// TIA Portal project "Sequential Tank Transfer System" (V17)

(* hardware
DEVICE "S7-1500/ET200MP station_1"  S7-1500 station
   slot 0: "Rail_0"  Rack  6ES7 590-1***0-0AA0
   slot 1: "PLC_STTS_01"  CPU 1512C-1 PN  6ES7 512-1CK00-0AB0  V2.9
      slot 3: "CPU display_1"  6ES7591-1AA00-0AA0
      slot 32768: "PROFINET interface_1"  X1
         slot 32769: "Port_1"  X1 P1
         slot 32770: "Port_2"  X1 P2
      slot 34817: "Virtual CP interface port_1"  Virtual CP interface port  Virtual CP interface port
DEVICE "HMI_1"  TP700 Comfort
   slot 0: "HMI_1"  TP700 Comfort  6AV2 124-0GC01-0AX0  17.0.0.0
   slot 1: "HMI_RT_1"  TP700 Comfort  6AV2 124-0GC01-0AX0  17.0.0.0
   slot 5: "HMI_1.IE_CP_1"  PROFINET Interface  17.0.0.0
      slot 1: "PROFINET Interface_1"  PROFINET Interface
         slot 1: "Port_1"  Port
         slot 2: "Port_2"  Port
   slot 7: "HMI_1.MPI/DP_CP_1"  MPI/DP Interface  17.0.0.0
*)

// ===== PLC "PLC_STTS_01"  CPU 1512C-1 PN =====

VAR_GLOBAL   // PLC tag table "STTS_Table"
   "PB_Start" AT %I10.0 : Bool;   // Begins the sequence
   "PB_Stop" AT %I10.1 : Bool;   // Emergency stop function
   "Max_Lvl_T1" AT %I10.2 : Bool;   // Indicates when Tank 1 is full
   "Min_Lvl_T1" AT %I10.3 : Bool;   // Indicates when Tank 1 is empty
   "Max_Lvl_T2" AT %I10.4 : Bool;   // Indicates when Tank 2 is full
   "Min_Lvl_T2" AT %I10.5 : Bool;   // Indicates when Tank 2 is empty
   "Is_Open_V1" AT %I10.6 : Bool;   // Confirmation that Valve 1 is fully open
   "Is_Closed_V1" AT %I10.7 : Bool;   // Confirmation that Valve 1 is fully closed
   "Is_Open_V2" AT %I11.0 : Bool;   // Confirmation that Valve 2 is fully open
   "Is_Closed_V2" AT %I11.1 : Bool;   // Confirmation that Valve 2 is fully closed
   "Is_Open_V3" AT %I11.2 : Bool;   // Confirmation that Valve 3 is fully open
   "Is_Closed_V3" AT %I11.3 : Bool;   // Confirmation that Valve 3 is fully closed
   "Is_Open_V4" AT %I11.4 : Bool;   // Confirmation that Valve 4 is fully open
   "Is_Closed_V4" AT %I11.5 : Bool;   // Confirmation that Valve 4 is fully closed
   "FBK_P2" AT %I11.6 : Bool;   // Running feedback from Pump 2
   "FBK_P3" AT %I11.7 : Bool;   // Running feedback from Pump 3
   "P2_in_Alarm" AT %I12.0 : Bool;   // Alarm status for Pump 2 - Indicates pump fault
   "P3_in_Alarm" AT %I12.1 : Bool;   // Alarm status for Pump 3 - Indicates pump fault
   "CMD_V1" AT %Q4.0 : Bool;   // Command to open/close Valve 1 - Controls flow to pit
   "CMD_V2" AT %Q4.1 : Bool;   // Command to open/close Valve 2 - Controls flow from Tank 1 to Tank 2
   "CMD_V3" AT %Q4.2 : Bool;   // Command to open/close Valve 3 - Controls flow from Tank 3
   "CMD_V4" AT %Q4.3 : Bool;   // Command to open/close Valve 4 - Controls flow to Tank 1
   "Start_P2" AT %Q4.4 : Bool;   // Starts Pump 2 - Transfers liquid from Tank 1 to Tank 2
   "Stop_P2" AT %Q4.5 : Bool;   // Stops Pump 2
   "Start_P3" AT %Q4.6 : Bool;   // Starts Pump 3 - Transfers liquid from Tank 3 to Tank 1
   "Stop_P3" AT %Q4.7 : Bool;   // Stops Pump 3
   "Cycle_Finished" AT %Q5.2 : Bool;   // Cycle is done after five discharges to the pit are made
   "Conditions_Met" AT %Q5.0 : Bool;   // All conditions are met and the system is ready
   "PB_Reset" AT %I12.2 : Bool;   // Resets the cycle once it is complete
   "Cycle_Started" AT %Q5.1 : Bool;   // Cycle has started running
   "Cycle_Reset" AT %Q5.3 : Bool;   // Cycle has been reset
END_VAR

DATA_BLOCK "System_Condition_Check_DB"   // DB5
{ S7_Optimized_Access := 'TRUE' }
VERSION : 0.1
// stored: InstanceOfName System_Condition_Check
"System_Condition_Check"
BEGIN
END_DATA_BLOCK

DATA_BLOCK "Tank1_Fill_DB"   // DB6
{ S7_Optimized_Access := 'TRUE' }
VERSION : 0.1
// stored: InstanceOfName Tank1_Fill
"Tank1_Fill"
BEGIN
END_DATA_BLOCK

DATA_BLOCK "Tank2_Fill_DB"   // DB7
{ S7_Optimized_Access := 'TRUE' }
VERSION : 0.1
// stored: InstanceOfName Tank2_Fill
"Tank2_Fill"
BEGIN
END_DATA_BLOCK

DATA_BLOCK "Main_Control_System_DB"   // DB8
{ S7_Optimized_Access := 'TRUE' }
VERSION : 0.1
// stored: InstanceOfName Main_Control_System
"Main_Control_System"
BEGIN
END_DATA_BLOCK

DATA_BLOCK "Discharge_DB"   // DB9
{ S7_Optimized_Access := 'TRUE' }
VERSION : 0.1
// stored: InstanceOfName Discharge
"Discharge"
BEGIN
END_DATA_BLOCK

DATA_BLOCK "Status_Reset_DB"   // DB10
{ S7_Optimized_Access := 'TRUE' }
VERSION : 0.1
// stored: InstanceOfName Status_Reset
"Status_Reset"
BEGIN
END_DATA_BLOCK

// folder: System blocks/Program resources

DATA_BLOCK "Fill_Timer_1_DB"   // DB2
{ S7_Optimized_Access := 'TRUE' }
AUTHOR : Simatic
FAMILY : IEC
NAME : IEC_TMR
VERSION : 1.0
// stored: InstanceOfName IEC_TIMER
"IEC_TIMER"
BEGIN
END_DATA_BLOCK

DATA_BLOCK "Fill_Timer_2_DB"   // DB3
{ S7_Optimized_Access := 'TRUE' }
AUTHOR : Simatic
FAMILY : IEC
NAME : IEC_TMR
VERSION : 1.0
// stored: InstanceOfName IEC_TIMER
"IEC_TIMER"
BEGIN
END_DATA_BLOCK

DATA_BLOCK "Discharge_Counter_DB"   // DB4
{ S7_Optimized_Access := 'TRUE' }
AUTHOR : Simatic
FAMILY : IEC
NAME : CNTR
VERSION : 1.0
// stored: InstanceOfName IEC_COUNTER
"IEC_COUNTER"
BEGIN
END_DATA_BLOCK

DATA_BLOCK "Discharge_Countdown_Timer_DB"   // DB12
{ S7_Optimized_Access := 'TRUE' }
AUTHOR : Simatic
FAMILY : IEC
NAME : IEC_TMR
VERSION : 1.0
// stored: InstanceOfName IEC_TIMER
"IEC_TIMER"
BEGIN
END_DATA_BLOCK

DATA_BLOCK "Discharge_Process_Timer_DB"   // DB13
{ S7_Optimized_Access := 'TRUE' }
AUTHOR : Simatic
FAMILY : IEC
NAME : IEC_TMR
VERSION : 1.0
// stored: InstanceOfName IEC_TIMER
"IEC_TIMER"
BEGIN
END_DATA_BLOCK

// folder: (top level)

FUNCTION_BLOCK "Main_Control_System"   // FB2, LAD
{ S7_Optimized_Access := 'TRUE' }
VERSION : 0.1
   VAR_INPUT
      Push_Button_Start : Bool;   // Begins the sequence
      Push_Button_Stop : Bool := false;   // Emergency stop function
      Push_Button_Reset : Bool;   // Resets the sequence once cycle is complete
   END_VAR
   VAR_OUTPUT
      Start : Bool;   // Starts the cycle
      Finish : Bool;   // Finshes the cycle after five discharges
      Reset : Bool;   // Resets the cycle after five discharges
   END_VAR
   VAR
      Actual_Step : Int;   // Checks the current state of the system
      Emergency_Stop : Bool;   // Emergency stop activated flag
      System_Ready : Bool;   // All conditions met to allow system start
      System_Running : Bool := false;   // Indicates that the sequence is actively running
      Discharge_Complete : Bool;   // Liquid finished discharging to pit
      HMI_Start_Command : Bool;   // Allows HMI to start the system
      HMI_Stop_Command : Bool;   // Allows HMI to stop the system
      HMI_Reset_Command : Bool;   // Allows HMI to reset the system once cycle is complete
      Emergency_Stop_Reset : Bool;   // Allows HMI to reset emergency status
      Close : Bool;   // Closes the valves and pumps
   END_VAR
   VAR_TEMP   // added for the SCL form of the ladder/FBD networks
      _w1 : Bool;
      _w2 : Bool;
   END_VAR
BEGIN

REGION Network 1: STATE 0: System Ready Check
   // Checks if the system is ready to activate
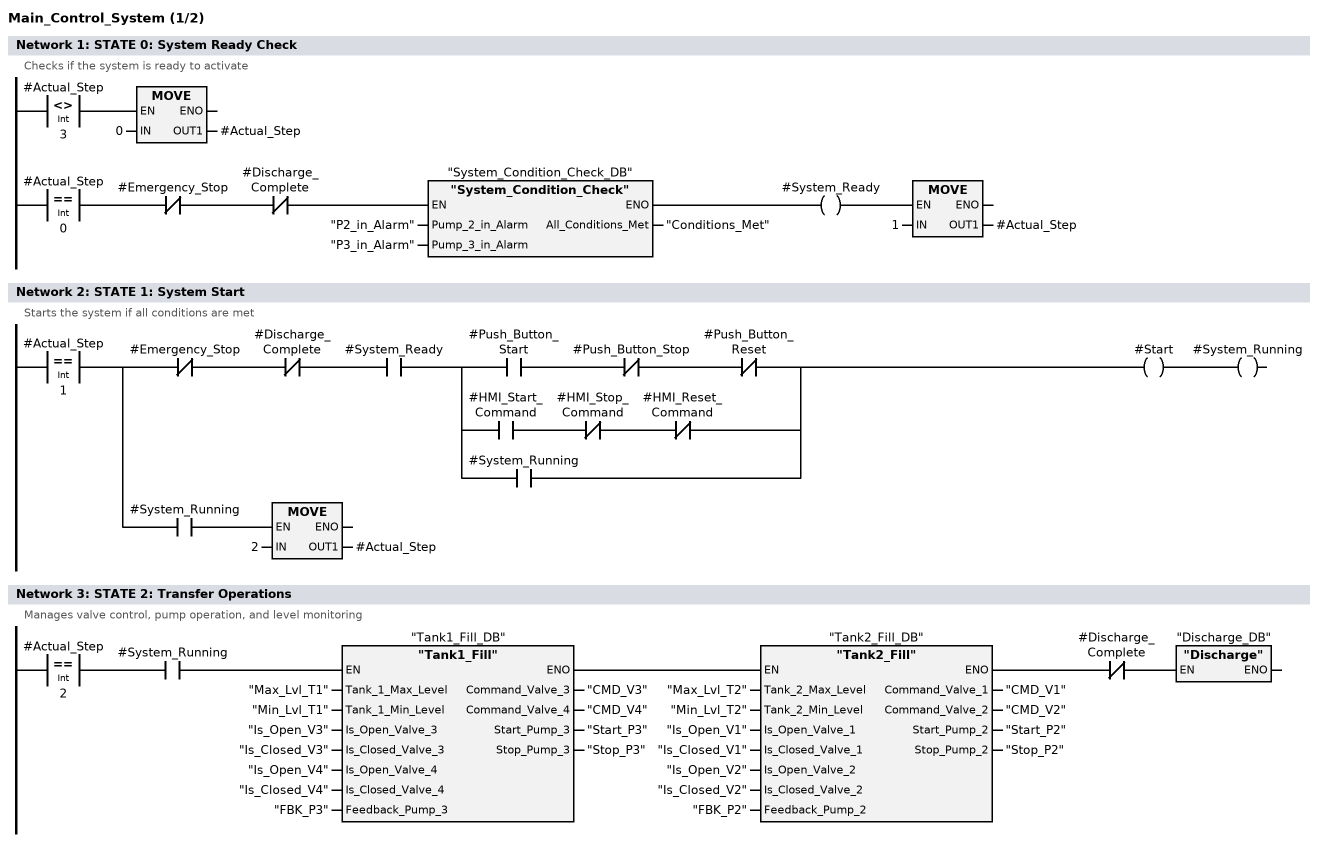
   RUNG wire#powerrail
      { S7_Templates := "SrcType := Int" } NE_Contact(in1 := #Actual_Step, in2 := 3)
      Move(in := 0, out1 => #Actual_Step)
   END_RUNG
   RUNG wire#powerrail
      { S7_Templates := "SrcType := Int" } EQ_Contact(in1 := #Actual_Step, in2 := 0)
      I_Contact( #Emergency_Stop )
      I_Contact( #Discharge_Complete )
      "System_Condition_Check_DB"(Pump_2_in_Alarm := "P2_in_Alarm", Pump_3_in_Alarm := "P3_in_Alarm", All_Conditions_Met => "Conditions_Met")
      Coil( #System_Ready )
      Move(in := 1, out1 => #Actual_Step)
   END_RUNG
   // the same network as SCL:
   IF #Actual_Step <> 3 THEN #Actual_Step := 0; END_IF;
   "System_Condition_Check_DB"(EN := (#Actual_Step = 0) AND NOT #Emergency_Stop AND NOT #Discharge_Complete,   // "System_Condition_Check"
                           Pump_2_in_Alarm := "P2_in_Alarm",
                           Pump_3_in_Alarm := "P3_in_Alarm",
                           All_Conditions_Met => "Conditions_Met",
                           ENO => #_w1);
   #System_Ready := #_w1;
   IF #_w1 THEN #Actual_Step := 1; END_IF;
END_REGION

REGION Network 2: STATE 1: System Start
   // Starts the system if all conditions are met
   RUNG wire#powerrail
      { S7_Templates := "SrcType := Int" } EQ_Contact(in1 := #Actual_Step, in2 := 1)
      wire#w1
      I_Contact( #Emergency_Stop )
      I_Contact( #Discharge_Complete )
      Contact( #System_Ready )
      wire#w2
      Contact( #Push_Button_Start )
      I_Contact( #Push_Button_Stop )
      I_Contact( #Push_Button_Reset )
      wire#w3
      Coil( #Start )
      Coil( #System_Running )
   END_RUNG
   RUNG wire#w2
      Contact( #HMI_Start_Command )
      I_Contact( #HMI_Stop_Command )
      I_Contact( #HMI_Reset_Command )
   END_RUNG wire#w3
   RUNG wire#w2
      Contact( #System_Running )
   END_RUNG wire#w3
   RUNG wire#w1
      Contact( #System_Running )
      Move(in := 2, out1 => #Actual_Step)
   END_RUNG
   // the same network as SCL:
   #_w1 := #Actual_Step = 1;
   #Start := #_w1 AND NOT #Emergency_Stop AND NOT #Discharge_Complete AND #System_Ready AND ((#Push_Button_Start AND NOT #Push_Button_Stop AND NOT #Push_Button_Reset) OR (#HMI_Start_Command AND NOT #HMI_Stop_Command AND NOT #HMI_Reset_Command) OR #System_Running);
   #System_Running := #Start;
   IF #_w1 AND #System_Running THEN #Actual_Step := 2; END_IF;
END_REGION

REGION Network 3: STATE 2: Transfer Operations
   // Manages valve control, pump operation, and level monitoring
   RUNG wire#powerrail
      { S7_Templates := "SrcType := Int" } EQ_Contact(in1 := #Actual_Step, in2 := 2)
      Contact( #System_Running )
      "Tank1_Fill_DB"(Tank_1_Max_Level := "Max_Lvl_T1", Tank_1_Min_Level := "Min_Lvl_T1", Is_Open_Valve_3 := "Is_Open_V3", Is_Closed_Valve_3 := "Is_Closed_V3", Is_Open_Valve_4 := "Is_Open_V4", Is_Closed_Valve_4 := "Is_Closed_V4", Feedback_Pump_3 := "FBK_P3", Command_Valve_3 => "CMD_V3", Command_Valve_4 => "CMD_V4", Start_Pump_3 => "Start_P3", Stop_Pump_3 => "Stop_P3")
      "Tank2_Fill_DB"(Tank_2_Max_Level := "Max_Lvl_T2", Tank_2_Min_Level := "Min_Lvl_T2", Is_Open_Valve_1 := "Is_Open_V1", Is_Closed_Valve_1 := "Is_Closed_V1", Is_Open_Valve_2 := "Is_Open_V2", Is_Closed_Valve_2 := "Is_Closed_V2", Feedback_Pump_2 := "FBK_P2", Command_Valve_1 => "CMD_V1", Command_Valve_2 => "CMD_V2", Start_Pump_2 => "Start_P2", Stop_Pump_2 => "Stop_P2")
      I_Contact( #Discharge_Complete )
      "Discharge_DB"()
   END_RUNG
   // the same network as SCL:
   "Tank1_Fill_DB"(EN := (#Actual_Step = 2) AND #System_Running,   // "Tank1_Fill"
                   Tank_1_Max_Level := "Max_Lvl_T1",
                   Tank_1_Min_Level := "Min_Lvl_T1",
                   Is_Open_Valve_3 := "Is_Open_V3",
                   Is_Closed_Valve_3 := "Is_Closed_V3",
                   Is_Open_Valve_4 := "Is_Open_V4",
                   Is_Closed_Valve_4 := "Is_Closed_V4",
                   Feedback_Pump_3 := "FBK_P3",
                   Command_Valve_3 => "CMD_V3",
                   Command_Valve_4 => "CMD_V4",
                   Start_Pump_3 => "Start_P3",
                   Stop_Pump_3 => "Stop_P3",
                   ENO => #_w1);
   "Tank2_Fill_DB"(EN := #_w1,   // "Tank2_Fill"
                   Tank_2_Max_Level := "Max_Lvl_T2",
                   Tank_2_Min_Level := "Min_Lvl_T2",
                   Is_Open_Valve_1 := "Is_Open_V1",
                   Is_Closed_Valve_1 := "Is_Closed_V1",
                   Is_Open_Valve_2 := "Is_Open_V2",
                   Is_Closed_Valve_2 := "Is_Closed_V2",
                   Feedback_Pump_2 := "FBK_P2",
                   Command_Valve_1 => "CMD_V1",
                   Command_Valve_2 => "CMD_V2",
                   Start_Pump_2 => "Start_P2",
                   Stop_Pump_2 => "Stop_P2",
                   ENO => #_w2);
   IF #_w2 AND NOT #Discharge_Complete THEN
       "Discharge_DB"();   // "Discharge"
   END_IF;
END_REGION

REGION Network 4: STATE 3: Finish and Reset Cycle
   // Finishes and resets the cycle after the liquid has been discharged to the pit no more than 5 times
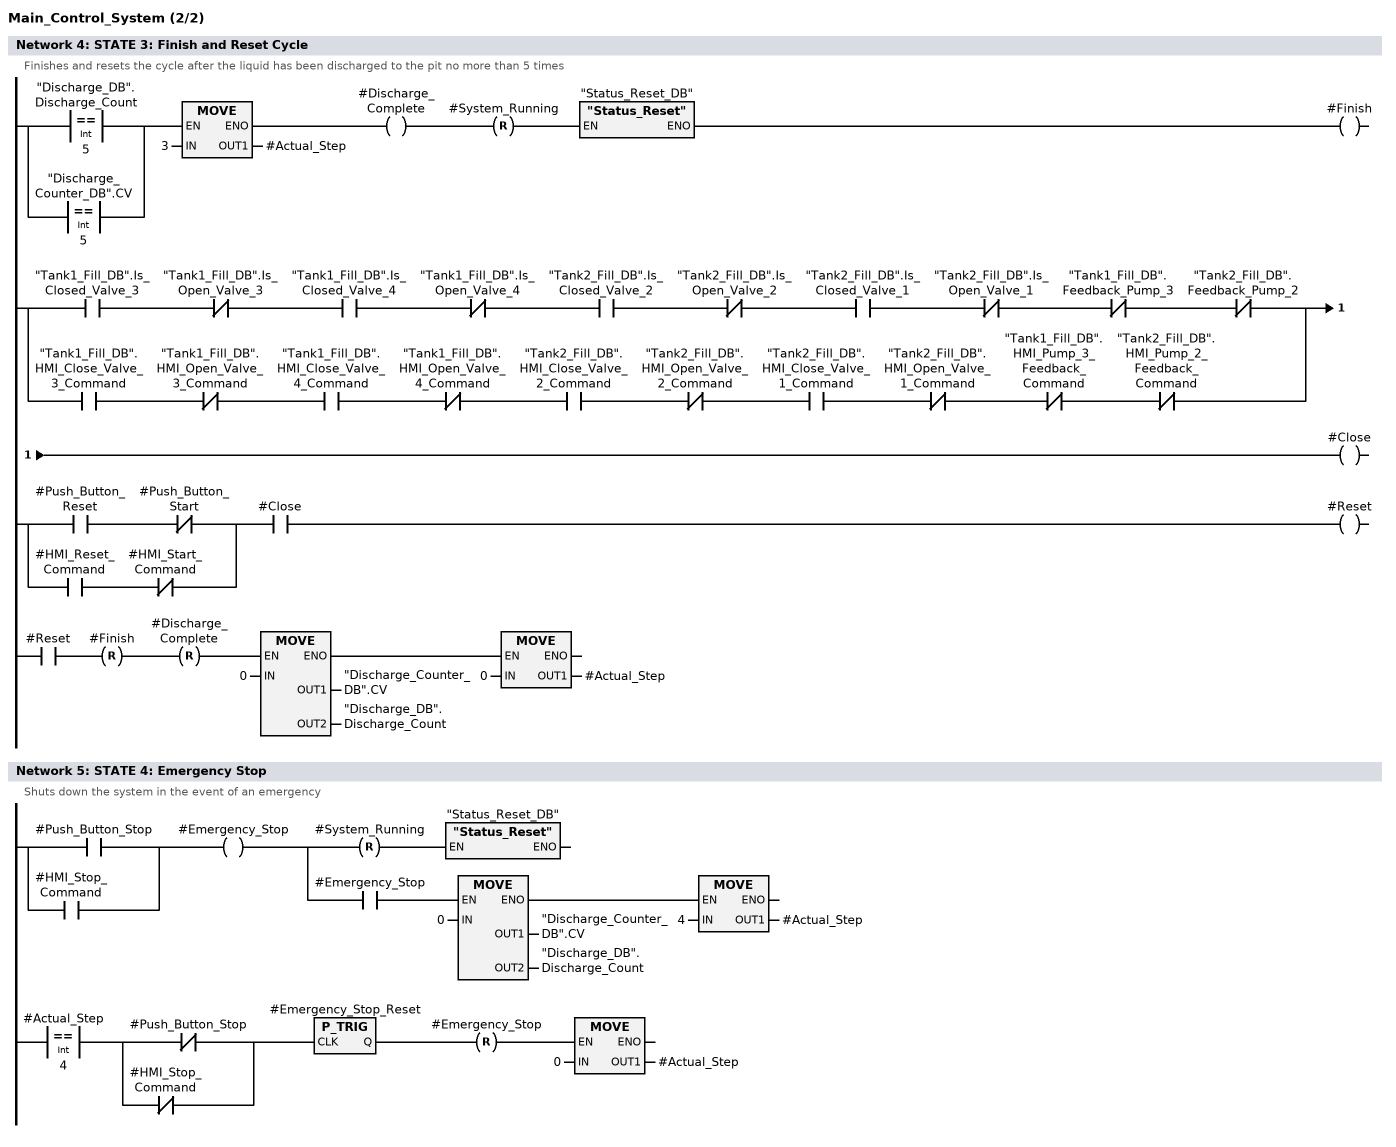
   RUNG wire#powerrail
      { S7_Templates := "SrcType := Int" } EQ_Contact(in1 := "Discharge_DB".Discharge_Count, in2 := 5)
      wire#w1
      Move(in := 3, out1 => #Actual_Step)
      Coil( #Discharge_Complete )
      R_Coil( #System_Running )
      "Status_Reset_DB"()
      Coil( #Finish )
   END_RUNG
   RUNG wire#powerrail
      { S7_Templates := "SrcType := Int" } EQ_Contact(in1 := "Discharge_Counter_DB".CV, in2 := 5)
   END_RUNG wire#w1
   RUNG wire#powerrail
      Contact( "Tank1_Fill_DB".Is_Closed_Valve_3 )
      I_Contact( "Tank1_Fill_DB".Is_Open_Valve_3 )
      Contact( "Tank1_Fill_DB".Is_Closed_Valve_4 )
      I_Contact( "Tank1_Fill_DB".Is_Open_Valve_4 )
      Contact( "Tank2_Fill_DB".Is_Closed_Valve_2 )
      I_Contact( "Tank2_Fill_DB".Is_Open_Valve_2 )
      Contact( "Tank2_Fill_DB".Is_Closed_Valve_1 )
      I_Contact( "Tank2_Fill_DB".Is_Open_Valve_1 )
      I_Contact( "Tank1_Fill_DB".Feedback_Pump_3 )
      I_Contact( "Tank2_Fill_DB".Feedback_Pump_2 )
      wire#w2
      Coil( #Close )
   END_RUNG
   RUNG wire#powerrail
      Contact( "Tank1_Fill_DB".HMI_Close_Valve_3_Command )
      I_Contact( "Tank1_Fill_DB".HMI_Open_Valve_3_Command )
      Contact( "Tank1_Fill_DB".HMI_Close_Valve_4_Command )
      I_Contact( "Tank1_Fill_DB".HMI_Open_Valve_4_Command )
      Contact( "Tank2_Fill_DB".HMI_Close_Valve_2_Command )
      I_Contact( "Tank2_Fill_DB".HMI_Open_Valve_2_Command )
      Contact( "Tank2_Fill_DB".HMI_Close_Valve_1_Command )
      I_Contact( "Tank2_Fill_DB".HMI_Open_Valve_1_Command )
      I_Contact( "Tank1_Fill_DB".HMI_Pump_3_Feedback_Command )
      I_Contact( "Tank2_Fill_DB".HMI_Pump_2_Feedback_Command )
   END_RUNG wire#w2
   RUNG wire#powerrail
      Contact( #Push_Button_Reset )
      I_Contact( #Push_Button_Start )
      wire#w3
      Contact( #Close )
      Coil( #Reset )
   END_RUNG
   RUNG wire#powerrail
      Contact( #HMI_Reset_Command )
      I_Contact( #HMI_Start_Command )
   END_RUNG wire#w3
   RUNG wire#powerrail
      Contact( #Reset )
      R_Coil( #Finish )
      R_Coil( #Discharge_Complete )
      Move(in := 0, out1 => "Discharge_Counter_DB".CV, out2 => "Discharge_DB".Discharge_Count)
      Move(in := 0, out1 => #Actual_Step)
   END_RUNG
   // the same network as SCL:
   #_w1 := ("Discharge_DB".Discharge_Count = 5) OR ("Discharge_Counter_DB".CV = 5);
   IF #_w1 THEN #Actual_Step := 3; END_IF;
   #Discharge_Complete := #_w1;
   IF #_w1 THEN #System_Running := FALSE; END_IF;
   "Status_Reset_DB"(EN := #_w1, ENO => #_w2);   // "Status_Reset"
   #Finish := #_w2;
   #Close := ("Tank1_Fill_DB".Is_Closed_Valve_3 AND NOT "Tank1_Fill_DB".Is_Open_Valve_3 AND "Tank1_Fill_DB".Is_Closed_Valve_4 AND NOT "Tank1_Fill_DB".Is_Open_Valve_4 AND "Tank2_Fill_DB".Is_Closed_Valve_2 AND NOT "Tank2_Fill_DB".Is_Open_Valve_2 AND "Tank2_Fill_DB".Is_Closed_Valve_1 AND NOT "Tank2_Fill_DB".Is_Open_Valve_1 AND NOT "Tank1_Fill_DB".Feedback_Pump_3 AND NOT "Tank2_Fill_DB".Feedback_Pump_2) OR ("Tank1_Fill_DB".HMI_Close_Valve_3_Command AND NOT "Tank1_Fill_DB".HMI_Open_Valve_3_Command AND "Tank1_Fill_DB".HMI_Close_Valve_4_Command AND NOT "Tank1_Fill_DB".HMI_Open_Valve_4_Command AND "Tank2_Fill_DB".HMI_Close_Valve_2_Command AND NOT "Tank2_Fill_DB".HMI_Open_Valve_2_Command AND "Tank2_Fill_DB".HMI_Close_Valve_1_Command AND NOT "Tank2_Fill_DB".HMI_Open_Valve_1_Command AND NOT "Tank1_Fill_DB".HMI_Pump_3_Feedback_Command AND NOT "Tank2_Fill_DB".HMI_Pump_2_Feedback_Command);
   #Reset := ((#Push_Button_Reset AND NOT #Push_Button_Start) OR (#HMI_Reset_Command AND NOT #HMI_Start_Command)) AND #Close;
   IF #Reset THEN
       #Finish := FALSE;
       #Discharge_Complete := FALSE;
       "Discharge_Counter_DB".CV := 0;
       "Discharge_DB".Discharge_Count := 0;
       #Actual_Step := 0;
   END_IF;
END_REGION

REGION Network 5: STATE 4: Emergency Stop
   // Shuts down the system in the event of an emergency
   RUNG wire#powerrail
      Contact( #Push_Button_Stop )
      wire#w1
      Coil( #Emergency_Stop )
      wire#w2
      R_Coil( #System_Running )
      "Status_Reset_DB"()
   END_RUNG
   RUNG wire#powerrail
      Contact( #HMI_Stop_Command )
   END_RUNG wire#w1
   RUNG wire#w2
      Contact( #Emergency_Stop )
      Move(in := 0, out1 => "Discharge_Counter_DB".CV, out2 => "Discharge_DB".Discharge_Count)
      Move(in := 4, out1 => #Actual_Step)
   END_RUNG
   RUNG wire#powerrail
      { S7_Templates := "SrcType := Int" } EQ_Contact(in1 := #Actual_Step, in2 := 4)
      wire#w3
      I_Contact( #Push_Button_Stop )
      wire#w4
      P_Trig( #Emergency_Stop_Reset )
      R_Coil( #Emergency_Stop )
      Move(in := 0, out1 => #Actual_Step)
   END_RUNG
   RUNG wire#w3
      I_Contact( #HMI_Stop_Command )
   END_RUNG wire#w4
   // the same network as SCL:
   #Emergency_Stop := #Push_Button_Stop OR #HMI_Stop_Command;
   IF #Emergency_Stop THEN
       #System_Running := FALSE;
       "Status_Reset_DB"();   // "Status_Reset"
   END_IF;
   IF #Emergency_Stop AND #Emergency_Stop THEN
       "Discharge_Counter_DB".CV := 0;
       "Discharge_DB".Discharge_Count := 0;
       #Actual_Step := 4;
   END_IF;
   #_w1 := (#Actual_Step = 4) AND (NOT #Push_Button_Stop OR NOT #HMI_Stop_Command);
   #_w2 := #_w1 AND NOT #Emergency_Stop_Reset;   // rising edge
   #Emergency_Stop_Reset := #_w1;
   IF #_w2 THEN
       #Emergency_Stop := FALSE;
       #Actual_Step := 0;
   END_IF;
END_REGION
END_FUNCTION_BLOCK

FUNCTION_BLOCK "System_Condition_Check"   // FB3, LAD
{ S7_Optimized_Access := 'TRUE' }
VERSION : 0.1
   VAR_INPUT
      Pump_2_in_Alarm : Bool;   // Alarm status for Pump 2 - Indicates pump fault
      Pump_3_in_Alarm : Bool;   // Alarm status for Pump 3 - Indicates pump fault
   END_VAR
   VAR_OUTPUT
      All_Conditions_Met : Bool;   // All conditions are met and the system is ready
   END_VAR
   VAR
      Valve_1_Status_OK : Bool;   // Valve 1 in known state
      Valve_2_Status_OK : Bool;   // Valve 2 in known state
      Valve_3_Status_OK : Bool;   // Valve 3 in known state
      Valve_4_Status_OK : Bool;   // Valve 4 in known state
      Tank_3_OK : Bool;
   END_VAR
   VAR CONSTANT
      Tank_3_Always_Full : Bool := True;   // Represents Tank 3's always-full status
   END_VAR
BEGIN

REGION Network 1: System Condition Check
   // Checks if all conditions are met before turning on the system
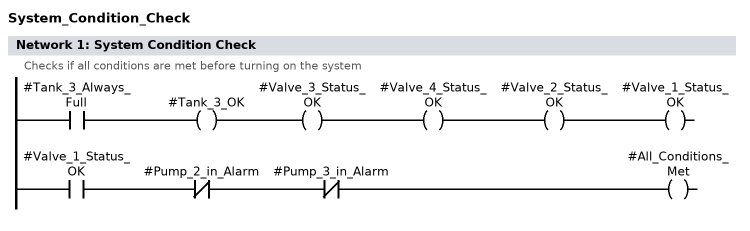
   RUNG wire#powerrail
      Contact( #Tank_3_Always_Full )
      Coil( #Tank_3_OK )
      Coil( #Valve_3_Status_OK )
      Coil( #Valve_4_Status_OK )
      Coil( #Valve_2_Status_OK )
      Coil( #Valve_1_Status_OK )
   END_RUNG
   RUNG wire#powerrail
      Contact( #Valve_1_Status_OK )
      I_Contact( #Pump_2_in_Alarm )
      I_Contact( #Pump_3_in_Alarm )
      Coil( #All_Conditions_Met )
   END_RUNG
   // the same network as SCL:
   #Tank_3_OK := #Tank_3_Always_Full;
   #Valve_3_Status_OK := #Tank_3_Always_Full;
   #Valve_4_Status_OK := #Tank_3_Always_Full;
   #Valve_2_Status_OK := #Tank_3_Always_Full;
   #Valve_1_Status_OK := #Tank_3_Always_Full;
   #All_Conditions_Met := #Valve_1_Status_OK AND NOT #Pump_2_in_Alarm AND NOT #Pump_3_in_Alarm;
END_REGION
END_FUNCTION_BLOCK

FUNCTION_BLOCK "Tank1_Fill"   // FB4, LAD
{ S7_Optimized_Access := 'TRUE' }
VERSION : 0.1
   VAR_INPUT
      Tank_1_Max_Level : Bool;   // Indicates when Tank 1 is full
      Tank_1_Min_Level : Bool;   // Indicates when Tank 1 is empty
      Is_Open_Valve_3 : Bool;   // Confirmation that Valve 3 is fully open
      Is_Closed_Valve_3 : Bool;   // Confirmation that Valve 3 is fully closed
      Is_Open_Valve_4 : Bool;   // Confirmation that Valve 4 is fully open
      Is_Closed_Valve_4 : Bool;   // Confirmation that Valve 4 is fully closed
      Feedback_Pump_3 : Bool;   // Running feedback from Pump 3
   END_VAR
   VAR_OUTPUT
      Command_Valve_3 : Bool;   // Command to open/close Valve 3 - Controls flow from Tank 3
      Command_Valve_4 : Bool;   // Command to open/close Valve 4 - Controls flow to Tank 1
      Start_Pump_3 : Bool;   // Command to start Pump 3 - Transfers liquid from Tank 3 to Tank 1
      Stop_Pump_3 : Bool;   // Command to stop Pump 3
   END_VAR
   VAR
      Tank_1_Fill_Active : Bool;   // Tank 1 currently filling
      Tank_1_Fill_Complete : Bool;   // Tank 1 has finished filling
      Tank_1_Fill_Preset_Time : Time := T#10s;   // Time set for Tank 1 filling
      Tank_1_Fill_Elapsed_Time : Time;   // Time it takes for Tank 1 to fill up
      Tank_1_Fill_Timer_Done : Bool;   // Timer for Tank 1 filling is done
      Tank_1_Fill_Seconds : Int;   // Allows HMI to read Tank 1 filling time
      HMI_Open_Valve_3_Command : Bool;   // Allows HMI to open Valve 3
      HMI_Close_Valve_3_Command : Bool;   // Allows HMI to close Valve 3
      HMI_Open_Valve_4_Command : Bool;   // Allows HMI to open Valve 4
      HMI_Close_Valve_4_Command : Bool;   // Allows HMI to close Valve 4
      HMI_Pump_3_Feedback_Command : Bool;   // Allows HMI to get running feedback from Pump 3
      Initialize_Tank_2 : Bool;   // Initiates Tank 2
      Initialize_Tank_1 : Bool;   // Initiates Tank 1
   END_VAR
   VAR_TEMP
      Tank_1_Fill_ET_DInt : DInt;
      Tank_1_Fill_ET_Div : DInt;
   END_VAR
   VAR_TEMP   // added for the SCL form of the ladder/FBD networks
      _w1 : Bool;
      _w2 : Bool;
      _w3 : Bool;
   END_VAR
BEGIN

REGION Network 1: Tank 1 Liquid Processing
   // Processes liquid from Tank 3 to Valve 3, Pump 3, and then Valve 4
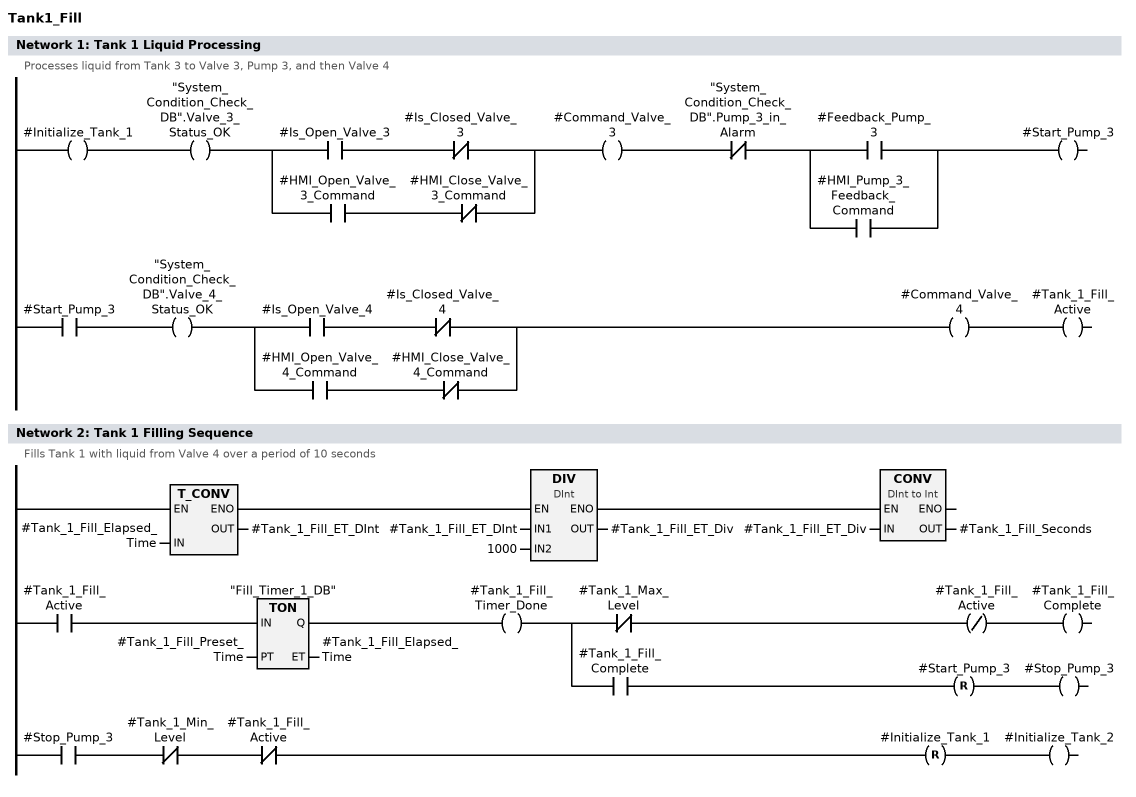
   RUNG wire#powerrail
      Coil( #Initialize_Tank_1 )
      Coil( "System_Condition_Check_DB".Valve_3_Status_OK )
      wire#w1
      Contact( #Is_Open_Valve_3 )
      I_Contact( #Is_Closed_Valve_3 )
      wire#w2
      Coil( #Command_Valve_3 )
      I_Contact( "System_Condition_Check_DB".Pump_3_in_Alarm )
      wire#w3
      Contact( #Feedback_Pump_3 )
      wire#w4
      Coil( #Start_Pump_3 )
   END_RUNG
   RUNG wire#w1
      Contact( #HMI_Open_Valve_3_Command )
      I_Contact( #HMI_Close_Valve_3_Command )
   END_RUNG wire#w2
   RUNG wire#w3
      Contact( #HMI_Pump_3_Feedback_Command )
   END_RUNG wire#w4
   RUNG wire#powerrail
      Contact( #Start_Pump_3 )
      Coil( "System_Condition_Check_DB".Valve_4_Status_OK )
      wire#w5
      Contact( #Is_Open_Valve_4 )
      I_Contact( #Is_Closed_Valve_4 )
      wire#w6
      Coil( #Command_Valve_4 )
      Coil( #Tank_1_Fill_Active )
   END_RUNG
   RUNG wire#w5
      Contact( #HMI_Open_Valve_4_Command )
      I_Contact( #HMI_Close_Valve_4_Command )
   END_RUNG wire#w6
   // the same network as SCL:
   #Initialize_Tank_1 := TRUE;
   "System_Condition_Check_DB".Valve_3_Status_OK := TRUE;
   #Command_Valve_3 := (#Is_Open_Valve_3 AND NOT #Is_Closed_Valve_3) OR (#HMI_Open_Valve_3_Command AND NOT #HMI_Close_Valve_3_Command);
   #Start_Pump_3 := #Command_Valve_3 AND NOT "System_Condition_Check_DB".Pump_3_in_Alarm AND (#Feedback_Pump_3 OR #HMI_Pump_3_Feedback_Command);
   "System_Condition_Check_DB".Valve_4_Status_OK := #Start_Pump_3;
   #Command_Valve_4 := #Start_Pump_3 AND ((#Is_Open_Valve_4 AND NOT #Is_Closed_Valve_4) OR (#HMI_Open_Valve_4_Command AND NOT #HMI_Close_Valve_4_Command));
   #Tank_1_Fill_Active := #Command_Valve_4;
END_REGION

REGION Network 2: Tank 1 Filling Sequence
   // Fills Tank 1 with liquid from Valve 4 over a period of 10 seconds
   // ENO of a box is taken as its EN; it also drops when the box reports an error
   #Tank_1_Fill_ET_DInt := T_CONV(IN := #Tank_1_Fill_Elapsed_Time);
   #Tank_1_Fill_ET_Div := #Tank_1_Fill_ET_DInt / 1000;
   #Tank_1_Fill_Seconds := DINT_TO_INT(#Tank_1_Fill_ET_Div);
   "Fill_Timer_1_DB".TON(IN := #Tank_1_Fill_Active,
                         PT := #Tank_1_Fill_Preset_Time,
                         ET => #Tank_1_Fill_Elapsed_Time);
   #Tank_1_Fill_Timer_Done := "Fill_Timer_1_DB".Q;
   #_w1 := "Fill_Timer_1_DB".Q AND NOT #Tank_1_Max_Level;
   #Tank_1_Fill_Active := NOT #_w1;
   #Tank_1_Fill_Complete := #_w1;
   #_w2 := "Fill_Timer_1_DB".Q AND #Tank_1_Fill_Complete;
   IF #_w2 THEN #Start_Pump_3 := FALSE; END_IF;
   #Stop_Pump_3 := #_w2;
   #_w3 := #Stop_Pump_3 AND NOT #Tank_1_Min_Level AND NOT #Tank_1_Fill_Active;
   IF #_w3 THEN #Initialize_Tank_1 := FALSE; END_IF;
   #Initialize_Tank_2 := #_w3;
END_REGION
END_FUNCTION_BLOCK

FUNCTION_BLOCK "Tank2_Fill"   // FB5, LAD
{ S7_Optimized_Access := 'TRUE' }
VERSION : 0.1
   VAR_INPUT
      Tank_2_Max_Level : Bool;   // Indicates when Tank 2 is full
      Tank_2_Min_Level : Bool;   // Indicates when Tank 2 is empty
      Is_Open_Valve_1 : Bool;   // Confirmation that Valve 1 is fully open
      Is_Closed_Valve_1 : Bool;   // Confirmation that Valve 1 is fully closed
      Is_Open_Valve_2 : Bool;   // Confirmation that Valve 2 is fully open
      Is_Closed_Valve_2 : Bool;   // Confirmation that Valve 2 is fully closed
      Feedback_Pump_2 : Bool;   // Running feedback from Pump 2
   END_VAR
   VAR_OUTPUT
      Command_Valve_1 : Bool;   // Command to open/close Valve 1 - Controls flow to pit
      Command_Valve_2 : Bool;   // Command to open/close Valve 2 - Controls flow from Tank 1 to Tank 2
      Start_Pump_2 : Bool;   // Command to start Pump 2 - Transfers liquid from Tank 1 to Tank 2
      Stop_Pump_2 : Bool;   // Command to stop Pump 2
   END_VAR
   VAR
      Tank_2_Fill_Active : Bool;   // Tank 2 currently filling
      Tank_2_Fill_Complete : Bool;   // Tank 2 has finished filling
      Tank_2_Fill_Preset_Time : Time := T#20s;   // Time set for Tank 2 filling
      Tank_2_Fill_Elapsed_Time : Time;   // Time it takes for Tank 2 to fill up
      Tank_2_Fill_Timer_Done : Bool;   // Timer for Tank 2 filling is done
      Tank_2_Fill_Seconds : Int;   // Allows HMI to read Tank 2 filling time
      Begin_Discharge_Countdown : Bool;   // Begins the countdown timer before the liquid can be discharged
      Discharge_Countdown_Preset_Time : Time := T#10s;   // Time set for discharge countdown
      Discharge_Countdown_Elapsed_Time : Time;   // Time it takes for discharge countdown to finish
      Discharge_Countdown_Seconds : Int;   // Allows HMI to read discharge countdown time
      Discharge_Countdown_Timer_Done : Bool;   // Timer for countdown to discharge is done
      Begin_Discharge : Bool;   // Begins discharging the liquid to the pit
      HMI_Open_Valve_1_Command : Bool;   // Allows HMI to open Valve 1
      HMI_Close_Valve_1_Command : Bool;   // Allows HMI to close Valve 1
      HMI_Open_Valve_2_Command : Bool;   // Allows HMI to open Valve 2
      HMI_Close_Valve_2_Command : Bool;   // Allows HMI to close Valve 2
      HMI_Pump_2_Feedback_Command : Bool;   // Allows HMI to get running feedback from Pump 2
   END_VAR
   VAR_TEMP
      Tank_2_Fill_ET_DInt : DInt;
      Tank_2_Fill_ET_Div : DInt;
      Discharge_Countdown_ET_DInt : DInt;
      Discharge_Countdown_ET_Div : DInt;
   END_VAR
   VAR_TEMP   // added for the SCL form of the ladder/FBD networks
      _w1 : Bool;
   END_VAR
BEGIN

REGION Network 1: Tank 2 Liquid Processing
   // Processes liquid from Tank 1 to Valve 2 and then Pump 2
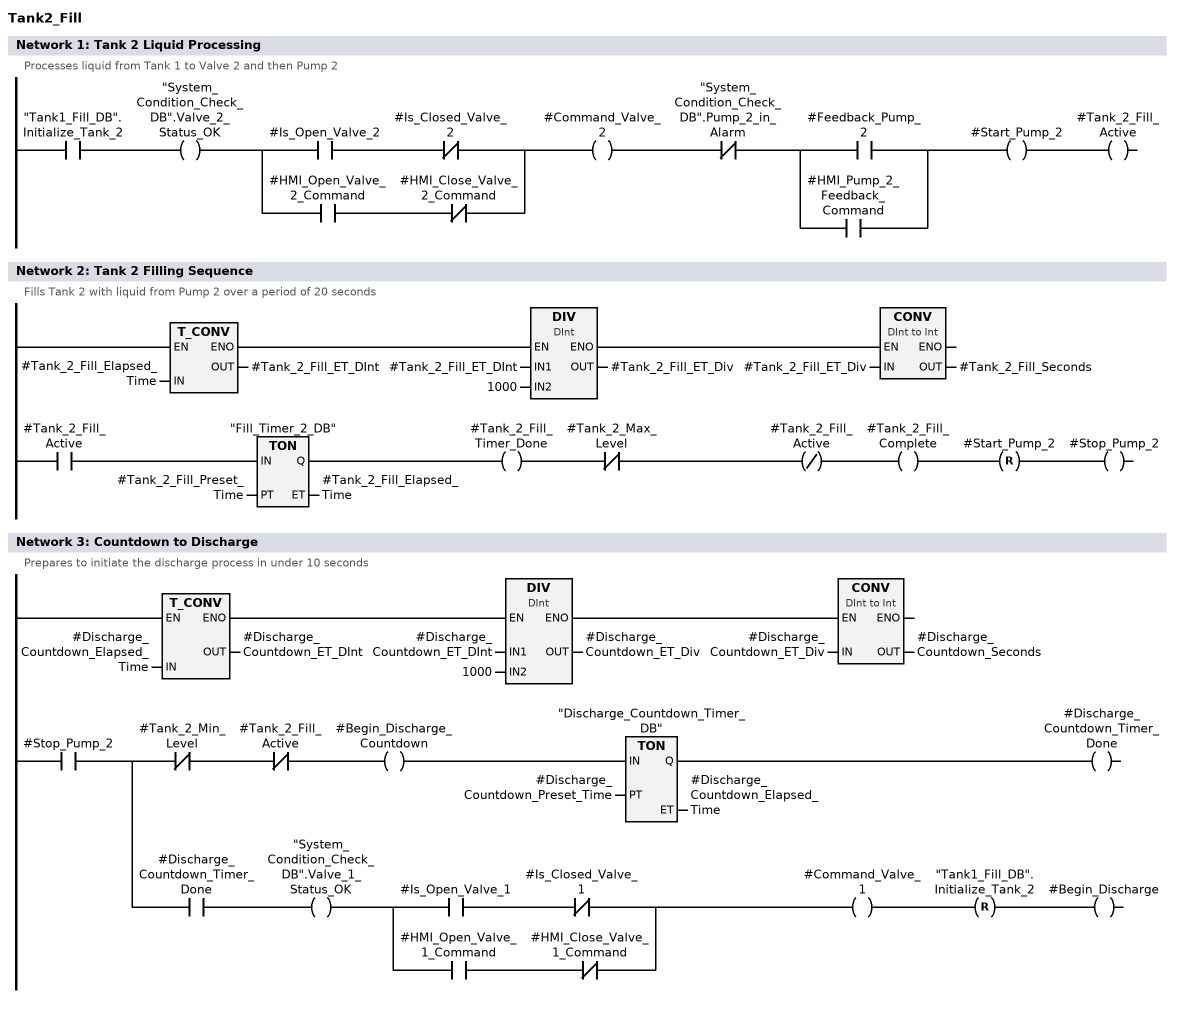
   RUNG wire#powerrail
      Contact( "Tank1_Fill_DB".Initialize_Tank_2 )
      Coil( "System_Condition_Check_DB".Valve_2_Status_OK )
      wire#w1
      Contact( #Is_Open_Valve_2 )
      I_Contact( #Is_Closed_Valve_2 )
      wire#w2
      Coil( #Command_Valve_2 )
      I_Contact( "System_Condition_Check_DB".Pump_2_in_Alarm )
      wire#w3
      Contact( #Feedback_Pump_2 )
      wire#w4
      Coil( #Start_Pump_2 )
      Coil( #Tank_2_Fill_Active )
   END_RUNG
   RUNG wire#w1
      Contact( #HMI_Open_Valve_2_Command )
      I_Contact( #HMI_Close_Valve_2_Command )
   END_RUNG wire#w2
   RUNG wire#w3
      Contact( #HMI_Pump_2_Feedback_Command )
   END_RUNG wire#w4
   // the same network as SCL:
   "System_Condition_Check_DB".Valve_2_Status_OK := "Tank1_Fill_DB".Initialize_Tank_2;
   #Command_Valve_2 := "Tank1_Fill_DB".Initialize_Tank_2 AND ((#Is_Open_Valve_2 AND NOT #Is_Closed_Valve_2) OR (#HMI_Open_Valve_2_Command AND NOT #HMI_Close_Valve_2_Command));
   #Start_Pump_2 := #Command_Valve_2 AND NOT "System_Condition_Check_DB".Pump_2_in_Alarm AND (#Feedback_Pump_2 OR #HMI_Pump_2_Feedback_Command);
   #Tank_2_Fill_Active := #Start_Pump_2;
END_REGION

REGION Network 2: Tank 2 Filling Sequence
   // Fills Tank 2 with liquid from Pump 2 over a period of 20 seconds
   // ENO of a box is taken as its EN; it also drops when the box reports an error
   #Tank_2_Fill_ET_DInt := T_CONV(IN := #Tank_2_Fill_Elapsed_Time);
   #Tank_2_Fill_ET_Div := #Tank_2_Fill_ET_DInt / 1000;
   #Tank_2_Fill_Seconds := DINT_TO_INT(#Tank_2_Fill_ET_Div);
   "Fill_Timer_2_DB".TON(IN := #Tank_2_Fill_Active,
                         PT := #Tank_2_Fill_Preset_Time,
                         ET => #Tank_2_Fill_Elapsed_Time);
   #Tank_2_Fill_Timer_Done := "Fill_Timer_2_DB".Q;
   #_w1 := "Fill_Timer_2_DB".Q AND NOT #Tank_2_Max_Level;
   #Tank_2_Fill_Active := NOT #_w1;
   #Tank_2_Fill_Complete := #_w1;
   IF #_w1 THEN #Start_Pump_2 := FALSE; END_IF;
   #Stop_Pump_2 := #_w1;
END_REGION

REGION Network 3: Countdown to Discharge
   // Prepares to initiate the discharge process in under 10 seconds
   // ENO of a box is taken as its EN; it also drops when the box reports an error
   #Discharge_Countdown_ET_DInt := T_CONV(IN := #Discharge_Countdown_Elapsed_Time);
   #Discharge_Countdown_ET_Div := #Discharge_Countdown_ET_DInt / 1000;
   #Discharge_Countdown_Seconds := DINT_TO_INT(#Discharge_Countdown_ET_Div);
   #Begin_Discharge_Countdown := #Stop_Pump_2 AND NOT #Tank_2_Min_Level AND NOT #Tank_2_Fill_Active;
   "Discharge_Countdown_Timer_DB".TON(IN := #Begin_Discharge_Countdown,
                           PT := #Discharge_Countdown_Preset_Time,
                           ET => #Discharge_Countdown_Elapsed_Time);
   #Discharge_Countdown_Timer_Done := "Discharge_Countdown_Timer_DB".Q;
   "System_Condition_Check_DB".Valve_1_Status_OK := #Stop_Pump_2 AND #Discharge_Countdown_Timer_Done;
   #Command_Valve_1 := "System_Condition_Check_DB".Valve_1_Status_OK AND ((#Is_Open_Valve_1 AND NOT #Is_Closed_Valve_1) OR (#HMI_Open_Valve_1_Command AND NOT #HMI_Close_Valve_1_Command));
   IF #Command_Valve_1 THEN "Tank1_Fill_DB".Initialize_Tank_2 := FALSE; END_IF;
   #Begin_Discharge := #Command_Valve_1;
END_REGION
END_FUNCTION_BLOCK

FUNCTION_BLOCK "Discharge"   // FB6, LAD
{ S7_Optimized_Access := 'TRUE' }
VERSION : 0.1
   VAR
      Discharge_Active : Bool;   // Liquid currently discharging to pit
      Counter_Reset : Bool := false;   // Resets the discharge counter
      Timer_OneShot : Bool;   // For discharge counting
      Discharge_Process_Preset_Time : Time := T#30s;   // Time set for discharge
      Discharge_Process_Elapsed_Time : Time;   // Time it takes for discharge to finish
      Discharge_Procces_Timer_Done : Bool;   // Timer for discharge is done
      Discharge_Process_Seconds : Int;   // Allows HMI to read discharge time
      Discharge_Limit : Int := 5;   // Max amount for how many times liquid discharges to pit
      Discharge_Count : Int;   // Tracks how many times liquid discharges to pit
   END_VAR
   VAR_TEMP
      Discharge_Process_ET_DInt : DInt;
      Discharge_Process_ET_Div : DInt;
   END_VAR
   VAR_TEMP   // added for the SCL form of the ladder/FBD networks
      _w1 : Bool;
      _w2 : Bool;
      _w3 : Bool;
   END_VAR
BEGIN

REGION Network 1: Liquid Discharge
   // Discharges the liqud to the pit
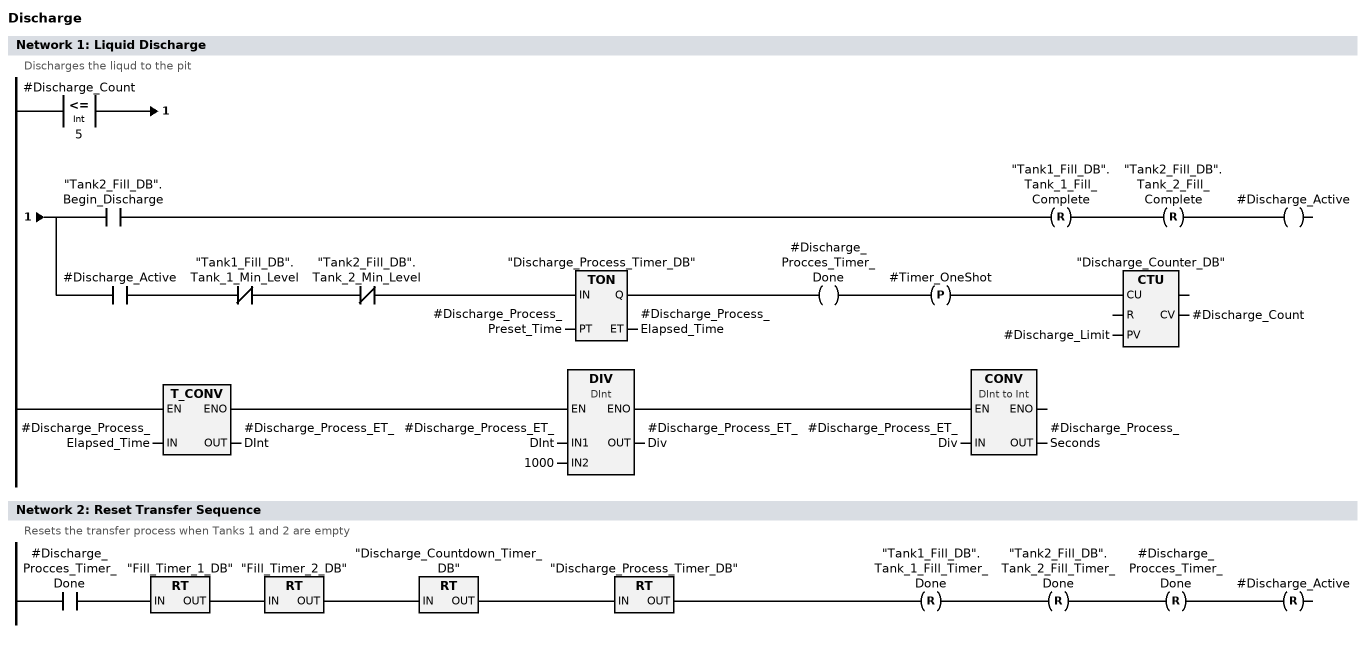
   // ENO of a box is taken as its EN; it also drops when the box reports an error
   #_w1 := #Discharge_Count <= 5;
   #_w2 := #_w1 AND "Tank2_Fill_DB".Begin_Discharge;
   IF #_w2 THEN
       "Tank1_Fill_DB".Tank_1_Fill_Complete := FALSE;
       "Tank2_Fill_DB".Tank_2_Fill_Complete := FALSE;
   END_IF;
   #Discharge_Active := #_w2;
   "Discharge_Process_Timer_DB".TON(IN := #_w1 AND #Discharge_Active AND NOT "Tank1_Fill_DB".Tank_1_Min_Level AND NOT "Tank2_Fill_DB".Tank_2_Min_Level,
                           PT := #Discharge_Process_Preset_Time,
                           ET => #Discharge_Process_Elapsed_Time);
   #Discharge_Procces_Timer_Done := "Discharge_Process_Timer_DB".Q;
   #_w3 := "Discharge_Process_Timer_DB".Q AND NOT #Timer_OneShot;   // rising edge
   #Timer_OneShot := "Discharge_Process_Timer_DB".Q;
   "Discharge_Counter_DB".CTU(CU := #_w3, PV := #Discharge_Limit, CV => #Discharge_Count);
   #Discharge_Process_ET_DInt := T_CONV(IN := #Discharge_Process_Elapsed_Time);
   #Discharge_Process_ET_Div := #Discharge_Process_ET_DInt / 1000;
   #Discharge_Process_Seconds := DINT_TO_INT(#Discharge_Process_ET_Div);
END_REGION

REGION Network 2: Reset Transfer Sequence
   // Resets the transfer process when Tanks 1 and 2 are empty
   RUNG wire#powerrail
      Contact( #Discharge_Procces_Timer_Done )
      RT_Coil( "Fill_Timer_1_DB" )
      RT_Coil( "Fill_Timer_2_DB" )
      RT_Coil( "Discharge_Countdown_Timer_DB" )
      RT_Coil( "Discharge_Process_Timer_DB" )
      R_Coil( "Tank1_Fill_DB".Tank_1_Fill_Timer_Done )
      R_Coil( "Tank2_Fill_DB".Tank_2_Fill_Timer_Done )
      R_Coil( #Discharge_Procces_Timer_Done )
      R_Coil( #Discharge_Active )
   END_RUNG
   // the same network as SCL:
   IF #Discharge_Procces_Timer_Done THEN
       RESET_TIMER("Fill_Timer_1_DB");
       RESET_TIMER("Fill_Timer_2_DB");
       RESET_TIMER("Discharge_Countdown_Timer_DB");
       RESET_TIMER("Discharge_Process_Timer_DB");
       "Tank1_Fill_DB".Tank_1_Fill_Timer_Done := FALSE;
       "Tank2_Fill_DB".Tank_2_Fill_Timer_Done := FALSE;
   END_IF;
   #_w1 := #Discharge_Procces_Timer_Done;
   IF #_w1 THEN
       #Discharge_Procces_Timer_Done := FALSE;
       #Discharge_Active := FALSE;
   END_IF;
END_REGION
END_FUNCTION_BLOCK

FUNCTION_BLOCK "Status_Reset"   // FB7, LAD
{ S7_Optimized_Access := 'TRUE' }
VERSION : 0.1
BEGIN

REGION Network 1: Status Reset
   // Resets the status of the valves, timers, tanks, and pumps
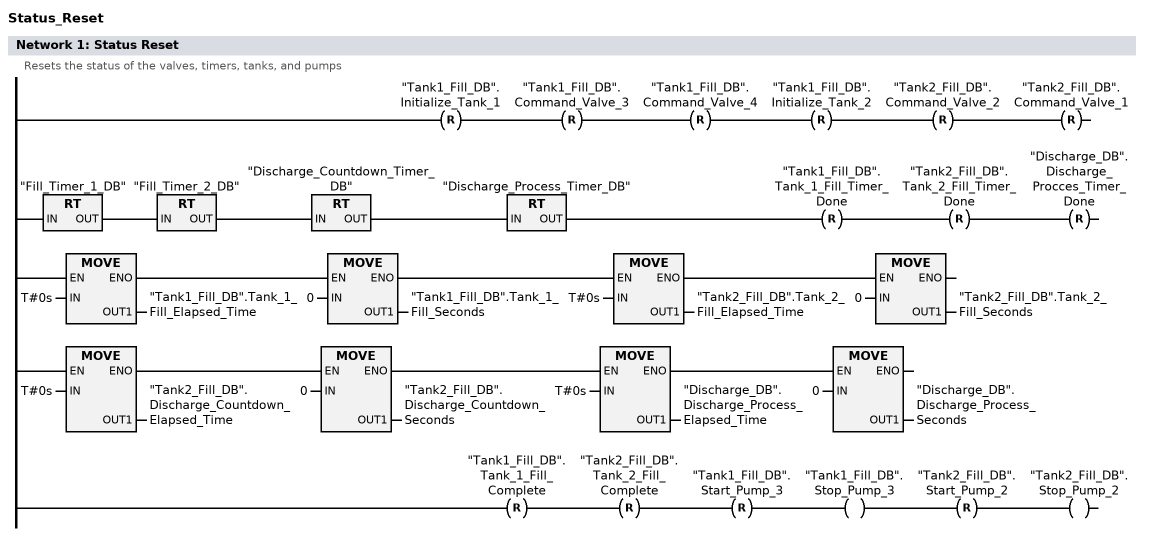
   RUNG wire#powerrail
      R_Coil( "Tank1_Fill_DB".Initialize_Tank_1 )
      R_Coil( "Tank1_Fill_DB".Command_Valve_3 )
      R_Coil( "Tank1_Fill_DB".Command_Valve_4 )
      R_Coil( "Tank1_Fill_DB".Initialize_Tank_2 )
      R_Coil( "Tank2_Fill_DB".Command_Valve_2 )
      R_Coil( "Tank2_Fill_DB".Command_Valve_1 )
   END_RUNG
   RUNG wire#powerrail
      RT_Coil( "Fill_Timer_1_DB" )
      RT_Coil( "Fill_Timer_2_DB" )
      RT_Coil( "Discharge_Countdown_Timer_DB" )
      RT_Coil( "Discharge_Process_Timer_DB" )
      R_Coil( "Tank1_Fill_DB".Tank_1_Fill_Timer_Done )
      R_Coil( "Tank2_Fill_DB".Tank_2_Fill_Timer_Done )
      R_Coil( "Discharge_DB".Discharge_Procces_Timer_Done )
   END_RUNG
   RUNG wire#powerrail
      Move(in := T#0s, out1 => "Tank1_Fill_DB".Tank_1_Fill_Elapsed_Time)
      Move(in := 0, out1 => "Tank1_Fill_DB".Tank_1_Fill_Seconds)
      Move(in := T#0s, out1 => "Tank2_Fill_DB".Tank_2_Fill_Elapsed_Time)
      Move(in := 0, out1 => "Tank2_Fill_DB".Tank_2_Fill_Seconds)
   END_RUNG
   RUNG wire#powerrail
      Move(in := T#0s, out1 => "Tank2_Fill_DB".Discharge_Countdown_Elapsed_Time)
      Move(in := 0, out1 => "Tank2_Fill_DB".Discharge_Countdown_Seconds)
      Move(in := T#0s, out1 => "Discharge_DB".Discharge_Process_Elapsed_Time)
      Move(in := 0, out1 => "Discharge_DB".Discharge_Process_Seconds)
   END_RUNG
   RUNG wire#powerrail
      R_Coil( "Tank1_Fill_DB".Tank_1_Fill_Complete )
      R_Coil( "Tank2_Fill_DB".Tank_2_Fill_Complete )
      R_Coil( "Tank1_Fill_DB".Start_Pump_3 )
      Coil( "Tank1_Fill_DB".Stop_Pump_3 )
      R_Coil( "Tank2_Fill_DB".Start_Pump_2 )
      Coil( "Tank2_Fill_DB".Stop_Pump_2 )
   END_RUNG
   // the same network as SCL:
   "Tank1_Fill_DB".Initialize_Tank_1 := FALSE;
   "Tank1_Fill_DB".Command_Valve_3 := FALSE;
   "Tank1_Fill_DB".Command_Valve_4 := FALSE;
   "Tank1_Fill_DB".Initialize_Tank_2 := FALSE;
   "Tank2_Fill_DB".Command_Valve_2 := FALSE;
   "Tank2_Fill_DB".Command_Valve_1 := FALSE;
   RESET_TIMER("Fill_Timer_1_DB");
   RESET_TIMER("Fill_Timer_2_DB");
   RESET_TIMER("Discharge_Countdown_Timer_DB");
   RESET_TIMER("Discharge_Process_Timer_DB");
   "Tank1_Fill_DB".Tank_1_Fill_Timer_Done := FALSE;
   "Tank2_Fill_DB".Tank_2_Fill_Timer_Done := FALSE;
   "Discharge_DB".Discharge_Procces_Timer_Done := FALSE;
   "Tank1_Fill_DB".Tank_1_Fill_Elapsed_Time := T#0s;
   "Tank1_Fill_DB".Tank_1_Fill_Seconds := 0;
   "Tank2_Fill_DB".Tank_2_Fill_Elapsed_Time := T#0s;
   "Tank2_Fill_DB".Tank_2_Fill_Seconds := 0;
   "Tank2_Fill_DB".Discharge_Countdown_Elapsed_Time := T#0s;
   "Tank2_Fill_DB".Discharge_Countdown_Seconds := 0;
   "Discharge_DB".Discharge_Process_Elapsed_Time := T#0s;
   "Discharge_DB".Discharge_Process_Seconds := 0;
   "Tank1_Fill_DB".Tank_1_Fill_Complete := FALSE;
   "Tank2_Fill_DB".Tank_2_Fill_Complete := FALSE;
   "Tank1_Fill_DB".Start_Pump_3 := FALSE;
   "Tank1_Fill_DB".Stop_Pump_3 := TRUE;
   "Tank2_Fill_DB".Start_Pump_2 := FALSE;
   "Tank2_Fill_DB".Stop_Pump_2 := TRUE;
END_REGION
END_FUNCTION_BLOCK

ORGANIZATION_BLOCK "Main"   // OB1, LAD, ProgramCycle
TITLE = "Main Program Sweep (Cycle)"
{ S7_Optimized_Access := 'TRUE' }
VERSION : 0.1
   VAR_INPUT
      Initial_Call : Bool;   // Initial call of this OB
      Remanence : Bool;   // =True, if remanent data are available
   END_VAR
BEGIN

REGION Network 1
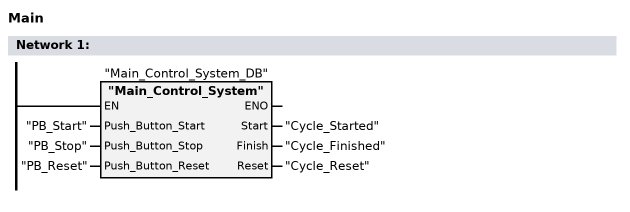
   RUNG wire#powerrail
      "Main_Control_System_DB"(Push_Button_Start := "PB_Start", Push_Button_Stop := "PB_Stop", Push_Button_Reset := "PB_Reset", Start => "Cycle_Started", Finish => "Cycle_Finished", Reset => "Cycle_Reset")
   END_RUNG
   // the same network as SCL:
   "Main_Control_System_DB"(Push_Button_Start := "PB_Start",   // "Main_Control_System"
                           Push_Button_Stop := "PB_Stop",
                           Push_Button_Reset := "PB_Reset",
                           Start => "Cycle_Started",
                           Finish => "Cycle_Finished",
                           Reset => "Cycle_Reset");
END_REGION
END_ORGANIZATION_BLOCK

(* ===== HMI "HMI_RT_1" =====
system functions are stored by id; their names below are inferred from use
connection "HMI_Connection_1": ETHERNET, S7_1500_OMS

HMI tags "STTS_HMI_Table"
   "Push_Button_Start" : Bool = PLC Main_Control_System_DB.HMI_Start_Command AT %DB1.DBX0.0, 100 ms
   "Push_Button_Stop" : Bool = PLC Main_Control_System_DB.HMI_Stop_Command AT %DB1.DBX0.0, 100 ms
   "System_Running" : Bool = PLC Main_Control_System_DB.System_Running AT %DB1.DBX0.0, 100 ms
   "Emergency_Stop" : Bool = PLC Main_Control_System_DB.Emergency_Stop AT %DB1.DBX0.0, 100 ms
   "System_Ready" : Bool = PLC Main_Control_System_DB.System_Ready AT %DB1.DBX0.0, 100 ms
   "Tank_3_Always_Full" : Bool = PLC System_Condition_Check_DB.Tank_3_OK AT %DB1.DBX0.0, 100 ms
   "Valve_3" : Bool = PLC Tank1_Fill_DB.Command_Valve_3 AT %DB1.DBX0.0, 100 ms
   "Valve_4" : Bool = PLC Tank1_Fill_DB.Command_Valve_4 AT %DB1.DBX0.0, 100 ms
   "Valve_2" : Bool = PLC Tank2_Fill_DB.Command_Valve_2 AT %DB1.DBX0.0, 100 ms
   "Valve_1" : Bool = PLC Tank2_Fill_DB.Command_Valve_1 AT %DB1.DBX0.0, 100 ms
   "Pump_3_Feedback" : Bool = PLC Tank1_Fill_DB.HMI_Pump_3_Feedback_Command AT %DB1.DBX0.0, 100 ms
   "Pump_2_Feedback" : Bool = PLC Tank2_Fill_DB.HMI_Pump_2_Feedback_Command AT %DB1.DBX0.0, 100 ms
   "Tank_1_Fill_Complete" : Bool = PLC Tank1_Fill_DB.Tank_1_Fill_Complete AT %DB1.DBX0.0, 100 ms
   "Tank_2_Fill_Complete" : Bool = PLC Tank2_Fill_DB.Tank_2_Fill_Complete AT %DB1.DBX0.0, 100 ms
   "Tank_1_Fill_Time" : Int = PLC Tank1_Fill_DB.Tank_1_Fill_Seconds AT %DB1.DBD0, 100 ms
   "Tank_2_Fill_Time" : Int = PLC Tank2_Fill_DB.Tank_2_Fill_Seconds AT %DB1.DBX0.0, 100 ms
   "Discharge_Time" : Int = PLC Discharge_DB.Discharge_Process_Seconds AT %DB1.DBD0, 100 ms
   "Discharge_Count" : Int = PLC Discharge_DB.Discharge_Count AT %DB1.DBW0, 100 ms
   "Finish" : Bool = PLC Main_Control_System_DB.Finish AT %DB1.DBX0.0, 100 ms
   "Push_Button_Reset" : Bool = PLC Main_Control_System_DB.HMI_Reset_Command AT %DB1.DBX0.0, 100 ms
   "Actual_Step" : Int = PLC Main_Control_System_DB.Actual_Step AT %DB1.DBX0.0, 100 ms
   "Discharge" : Bool = PLC Discharge_DB.Discharge_Active AT %DB1.DBW0, 100 ms
   "Discharge_Countdown" : Int = PLC Tank2_Fill_DB.Discharge_Countdown_Seconds AT %DB1.DBX0.0, 100 ms
   "Open_Valve_3" : Bool = PLC Tank1_Fill_DB.HMI_Open_Valve_3_Command AT %DB1.DBX0.0, 100 ms
   "Open_Valve_4" : Bool = PLC Tank1_Fill_DB.HMI_Open_Valve_4_Command AT %DB1.DBX0.0, 100 ms
   "Close_Valve_3" : Bool = PLC Tank1_Fill_DB.HMI_Close_Valve_3_Command AT %DB1.DBX0.0, 100 ms
   "Close_Valve_4" : Bool = PLC Tank1_Fill_DB.HMI_Close_Valve_4_Command AT %DB1.DBX0.0, 100 ms
   "Start_Pump_3" : Bool = PLC Tank1_Fill_DB.Start_Pump_3 AT %DB1.DBX0.0, 100 ms
   "Stop_Pump_3" : Bool = PLC Tank1_Fill_DB.Stop_Pump_3 AT %DB1.DBX0.0, 100 ms
   "Stop_Pump_2" : Bool = PLC Tank2_Fill_DB.Stop_Pump_2 AT %DB1.DBX0.0, 100 ms
   "Open_Valve_1" : Bool = PLC Tank2_Fill_DB.HMI_Open_Valve_1_Command AT %DB1.DBX0.0, 100 ms
   "Open_Valve_2" : Bool = PLC Tank2_Fill_DB.HMI_Open_Valve_2_Command AT %DB1.DBX0.0, 100 ms
   "Close_Valve_1" : Bool = PLC Tank2_Fill_DB.HMI_Close_Valve_1_Command AT %DB1.DBX0.0, 100 ms
   "Close_Valve_2" : Bool = PLC Tank2_Fill_DB.HMI_Close_Valve_2_Command AT %DB1.DBX0.0, 100 ms
   "Start_Pump_2" : Bool = PLC Tank2_Fill_DB.Start_Pump_2 AT %DB1.DBX0.0, 100 ms

screen "System_Screen" 800x480
   GraphicIOField "System_Running_LED" at 29,391 size 50x50; PictureOn "PilotLight_Square_G_On_256c"; PictureOff "PilotLight_Square_G_Off_256c"
      ProcessValue <- "System_Running"
   GraphicIOField "Emergency_Stop_LED" at 130,391 size 50x50; PictureOn "PilotLight_Square_R_On_256c"; PictureOff "PilotLight_Square_R_Off_256c"
      ProcessValue <- "Emergency_Stop"
   Rectangle "Tank_1" at 318,18 size 150x150
      Appearance <- "Tank_1_Fill_Complete"
   Rectangle "Tank_2" at 634,179 size 150x150
      Appearance <- "Tank_2_Fill_Complete"
   Rectangle "Tank_3" at 10,178 size 150x150
      Appearance <- "Tank_3_Always_Full"
   Polyline "Pipe_1" at 159,166 size 241x147
      Appearance <- "System_Ready"
   Circle "Pump_3" at 330,284 size 48x48
      Appearance <- "Pump_3_Feedback"
   Polyline "Pipe_2" at 467,145 size 254x36
      Appearance <- "System_Ready"
   Circle "Pump_2" at 632,119 size 48x48
      Appearance <- "Pump_2_Feedback"
   Line "Pipe_3" at 710,328 size 3x117
      Appearance <- "System_Ready"
   Polygon "Valve_3" at 216,297 size 69x31
      Appearance <- "Valve_3"
   Polygon "Valve_1" at 696,351 size 31x69
      Appearance <- "Valve_1"
   Polygon "Valve_2" at 515,131 size 69x31
      Appearance <- "Valve_2"
   Polygon "Valve_4" at 383,185 size 31x69
      Appearance <- "Valve_4"
   Button "Start_Button" at 6,351 size 96x32; TextOff 'Start'
      on Press: InvertBit("Push_Button_Start")
   Button "Stop_Button" at 110,351 size 96x32; TextOff 'Stop'
      on Press: InvertBit("Push_Button_Stop")
   IOField "I/O field_1" at 147,39 size 90x32; FormatPattern 99; Unit  s
      ProcessValue <- "Tank_1_Fill_Time"
   IOField "I/O field_2" at 461,216 size 92x32; FormatPattern 99; Unit  s
      ProcessValue <- "Tank_2_Fill_Time"
   IOField "I/O field_3" at 506,365 size 80x32; FormatPattern 99; Unit  s
      ProcessValue <- "Discharge_Time"
   Polyline "Pit" at 655,444 size 128x24
      Appearance <- "Discharge"
   TextField "Text field_1" at 147,10 size 170x30; Text 'Tank 1 Fill Time'
   TextField "Text field_2" at 462,185 size 170x30; Text 'Tank 2 Fill Time'
   TextField "Text field_3" at 504,335 size 170x30; Text 'Discharge Time'
   TextField "Text field_4" at 204,265 size 90x30; Text 'Valve 3'
   TextField "Text field_5" at 307,253 size 90x30; Text 'Pump 3'
   TextField "Text field_6" at 299,207 size 90x30; Text 'Valve 4'
   TextField "Text field_7" at 511,98 size 90x30; Text 'Valve 2'
   TextField "Text field_8" at 612,87 size 90x30; Text 'Pump 2'
   TextField "Text field_9" at 608,369 size 90x30; Text 'Valve 1'
   TextField "Text field_10" at 30,145 size 100x30; Text 'Tank 3'
   TextField "Text field_11" at 471,4 size 100x30; Text 'Tank 1'
   TextField "Text field_12" at 721,145 size 75x30; Text 'Tank 2'
   TextField "Text field_13" at 602,445 size 50x30; Text 'Pit'
   TextField "Text field_14" at 162,313 size 50x30; Text 'OUT'
   TextField "Text field_15" at 354,166 size 45x30; Text 'IN'
   TextField "Text field_16" at 466,115 size 50x30; Text 'OUT'
   TextField "Text field_17" at 694,153 size 45x30; Text 'IN'
   TextField "Text field_18" at 727,329 size 50x30; Text 'OUT'
   IOField "I/O field_4" at 499,436 size 85x32; FormatPattern 9
      ProcessValue <- "Discharge_Count"
   TextField "Text field_19" at 496,403 size 175x30; Text 'Discharge Count'
   GraphicIOField "Finish_LED" at 235,391 size 50x50; PictureOn "PilotLight_Square_GN_On_256c"; PictureOff "PilotLight_Square_GN_Off_256c"
      ProcessValue <- "Finish"
   Button "Reset_Button" at 212,351 size 96x32; TextOff 'Reset'
      on Press: InvertBit("Push_Button_Reset")
   IOField "I/O field_5" at 7,39 size 55x32; FormatPattern 9
      ProcessValue <- "Actual_Step"
   TextField "Text field_20" at 7,9 size 140x30; Text 'Actual Step'
   IOField "I/O field_6" at 406,293 size 113x32; FormatPattern 99; Unit  s
      ProcessValue <- "Discharge_Countdown"
   TextField "Text field_21" at 405,258 size 225x30; Text 'Discharge Countdown'
   Button "Pump_3_Feedback_Button" at 325,351 size 160x32; TextOff 'Pump 3 Feedback'
      on Press: InvertBit("Pump_3_Feedback")
   Rectangle "Valve_3_Close_Sensor" at 291,302 size 4x23
      Appearance <- "Close_Valve_3"
   Rectangle "Valve_3_Open_Sensor" at 205,302 size 4x23
      Appearance <- "Open_Valve_3"
   Rectangle "Pump_3_Stop_Sensor" at 382,302 size 4x23
      Appearance <- "Stop_Pump_3"
   Rectangle "Pump_3_Start_Sensor" at 321,302 size 4x23
      Appearance <- "Start_Pump_3"
   Rectangle "Valve_4_Open_Sensor" at 389,260 size 23x4
      Appearance <- "Open_Valve_4"
   Rectangle "Valve_4_Close_Sensor" at 389,174 size 23x4
      Appearance <- "Close_Valve_4"
   Rectangle "Valve_2_Open_Sensor" at 504,135 size 4x23
      Appearance <- "Open_Valve_2"
   Rectangle "Valve_2_Close_Sensor" at 592,135 size 4x23
      Appearance <- "Close_Valve_2"
   Rectangle "Pump_2_Start_Sensor" at 618,135 size 4x23
      Appearance <- "Start_Pump_2"
   Rectangle "Pump_2_Stop_Sensor" at 685,135 size 4x23
      Appearance <- "Stop_Pump_2"
   Rectangle "Valve_1_Open_Sensor" at 699,339 size 23x4
      Appearance <- "Open_Valve_1"
   Rectangle "Valve_1_Close_Sensor" at 699,429 size 23x4
      Appearance <- "Close_Valve_1"
   Button "Pump_2_Feedback_Button" at 325,409 size 160x32; TextOff 'Pump 2 Feedback'
      on Press: InvertBit("Pump_2_Feedback")
   Switch "Valve_3_Switch" at 6,79 size 129x54; CaptionText 'Valve 3 Switch'; TextOff 'CLOSE'; TextOn 'OPEN'
      on SwitchOn: SetBit("Open_Valve_3"); ResetBit("Close_Valve_3")
      on SwitchOff: SetBit("Close_Valve_3"); ResetBit("Open_Valve_3")
      ProcessValue <- "Open_Valve_3"
   Switch "Valve_4_Switch" at 180,79 size 129x54; TextOn 'OPEN'; CaptionText 'Valve 4 Switch'; TextOff 'CLOSE'
      on SwitchOff: SetBit("Close_Valve_4"); ResetBit("Open_Valve_4")
      on SwitchOn: SetBit("Open_Valve_4"); ResetBit("Close_Valve_4")
      ProcessValue <- "Open_Valve_4"
   Switch "Valve_2_Switch" at 483,33 size 129x54; TextOn 'OPEN'; CaptionText 'Valve 2 Switch'; TextOff 'CLOSE'
      on SwitchOff: SetBit("Close_Valve_2"); ResetBit("Open_Valve_2")
      on SwitchOn: SetBit("Open_Valve_2"); ResetBit("Close_Valve_2")
      ProcessValue <- "Open_Valve_2"
   Switch "Valve_1_Switch" at 660,33 size 129x54; TextOn 'OPEN'; CaptionText 'Valve 1 Switch'; TextOff 'CLOSE'
      on SwitchOff: SetBit("Close_Valve_1"); ResetBit("Open_Valve_1")
      on SwitchOn: SetBit("Open_Valve_1"); ResetBit("Close_Valve_1")
      ProcessValue <- "Open_Valve_1"
*)